// TwinCAT 3 PLC project Main
// ProgramVersion: 3.1.4024.0
// libraries:
//   Tc2_Standard, * (Beckhoff Automation GmbH)
//   Tc2_System, * (Beckhoff Automation GmbH)
//   Tc3_Module, * (Beckhoff Automation GmbH)
// project tree:
//   GVLs/ GVL.TcGVL
//   / PlcTask.TcTTO
//   POUs/Devices/Light/ I_LIGHT.TcIO, Light.TcPOU
//   POUs/Devices/OperatorPanel/ SlitterMainOperatorPanel.TcPOU
//   POUs/Devices/PushButton/ I_PushButton.TcIO, NormallyClosePushButton.TcPOU, NormallyOpenPushButton.TcPOU
//   POUs/ MAIN.TcPOU
// real-time tasks:
//   TASK PlcTask: cycle T#10ms, priority 20, ADS port 350

CONFIGURATION Main
    RESOURCE PLC ON TwinCAT3
        TASK PlcTask(INTERVAL := T#10ms, PRIORITY := 20);
        PROGRAM MAIN WITH PlcTask : MAIN;
    END_RESOURCE
END_CONFIGURATION

// ---- GVLs/GVL.TcGVL
{attribute 'qualified_only'}
VAR_GLOBAL
	
	MainPanel		:	SlitterMainOperatorPanel();//(StartPB, StopPB, StartLight, StopLight);

END_VAR

// ---- POUs/Devices/Light/I_LIGHT.TcIO
INTERFACE I_LIGHT

METHOD Off
VAR_INPUT
END_VAR
END_METHOD

METHOD On
VAR_INPUT
END_VAR
END_METHOD

END_INTERFACE

// ---- POUs/Devices/PushButton/I_PushButton.TcIO
INTERFACE I_PushButton

PROPERTY IsPressed : BOOL
GET
END_GET
END_PROPERTY

PROPERTY IsReleased : BOOL
GET
END_GET
END_PROPERTY

END_INTERFACE

// ---- POUs/MAIN.TcPOU
PROGRAM MAIN
VAR
	Test	:	BOOL;
END_VAR

IF GVL.MainPanel.StopPressed THEN
	
	GVL.MainPanel.StopLightOn();
	GVL.MainPanel.StartLightOff();

ELSIF GVL.MainPanel.StartPressed AND GVL.MainPanel.StopReleased THEN

	GVL.MainPanel.StopLightOff();
	GVL.MainPanel.StartLightOn();	

END_IF

END_PROGRAM

// ---- POUs/Devices/OperatorPanel/SlitterMainOperatorPanel.TcPOU
{attribute 'monitoring':='call'}
FUNCTION_BLOCK SlitterMainOperatorPanel

VAR
	
	StartPB		:		NormallyOpenPushButton;
	StopPB		:		NormallyClosePushButton;
	
	StartLight	:		Light;
	StopLight	:		Light;

END_VAR

METHOD PUBLIC StartLightOff : BOOL
VAR_INPUT
END_VAR
StartLight.Off();
END_METHOD

METHOD PUBLIC StartLightOn : BOOL
VAR_INPUT
END_VAR
StartLight.On();
END_METHOD

PROPERTY PUBLIC StartPressed : Bool
GET
StartPressed := StartPB;
END_GET
END_PROPERTY

PROPERTY PUBLIC StartReleased : Bool
GET
StartReleased := NOT StartPressed;
END_GET
END_PROPERTY

METHOD PUBLIC StopLightOff : BOOL
VAR_INPUT
END_VAR
StopLight.Off();
END_METHOD

METHOD PUBLIC StopLightOn : BOOL
VAR_INPUT
END_VAR
StopLight.On();
END_METHOD

PROPERTY PUBLIC StopPressed : Bool
GET
StopPressed := Not StopPB;
END_GET
END_PROPERTY

PROPERTY PUBLIC StopReleased : Bool
GET
StopPressed := Not StopPressed;
END_GET
END_PROPERTY

END_FUNCTION_BLOCK

// ---- POUs/Devices/PushButton/NormallyOpenPushButton.TcPOU
FUNCTION_BLOCK NormallyOpenPushButton IMPLEMENTS I_PushButton

VAR
	Input	AT %I* : BOOL; 
END_VAR

PROPERTY IsPressed : BOOL
GET
IsPressed := Input;
END_GET
END_PROPERTY

PROPERTY IsReleased : BOOL
GET
IsReleased := NOT IsPressed;
END_GET
END_PROPERTY

END_FUNCTION_BLOCK

// ---- POUs/Devices/PushButton/NormallyClosePushButton.TcPOU
FUNCTION_BLOCK NormallyClosePushButton IMPLEMENTS I_PushButton

VAR
	Input	AT %I* : BOOL; 
END_VAR

PROPERTY IsPressed : BOOL
GET
IsPressed := NOT Input;
END_GET
END_PROPERTY

PROPERTY IsReleased : BOOL
GET
IsReleased := NOT IsPressed;
END_GET
END_PROPERTY

END_FUNCTION_BLOCK

// ---- POUs/Devices/Light/Light.TcPOU
FUNCTION_BLOCK Light IMPLEMENTS I_LIGHT

VAR
	Output AT %Q* : BOOL;
END_VAR

METHOD Off
Output := FALSE;
END_METHOD

METHOD On
Output := TRUE;
END_METHOD

END_FUNCTION_BLOCK
